(* Logix 5000 project; controller Leitura_AlfaInstrumentos_2711 vendor 1 type 14 code 149 rev 20.19; software revision 20.04 *)

TASK MainTask (continuous, watchdog 500 ms) : Balancas

MODULES
   Local : vendor 1 type 14 code 149 (Compact 0, rev 20.19)
      Discrete_IO : Embedded (Compact 1, rev 3.1, Output RPI 20 ms)
      BL04 : vendor 90 type 0 code 46 (Ethernet 192.168.1.53, rev 1.5, StandardDataDriven RPI 10 ms)
           BL04:I.DATA[5].1   // Unidade
           BL04:I.DATA[5].5   // 1 = Vazia
           BL04:I.DATA[5].0   // 1 = Erro
           BL04:I.DATA[15]   // Tara
           BL04:I.DATA[14]   // Tara
           BL04:I.DATA[13]   // Tara
           BL04:I.DATA[12]   // Tara
           BL04:I.DATA[5].2   // Unidade
           BL04:I.DATA[10]   // Peso Bruto ou Liquido
           BL04:I.DATA[8]   // Peso Bruto ou Liquido
           BL04:I.DATA[9]   // Peso Bruto ou Liquido
           BL04:I.DATA[11]   // Peso Bruto ou Liquido
           BL04:I.DATA[4].7   // 0 = Peso Bruto / 1 = Peso Liquido
           BL04:I.DATA[4].0   // Casas Decimais
           BL04:I.DATA[4].1   // Casas Decimais
           BL04:I.DATA[4].2   // Casas Decimais
           BL04:I.DATA[5].6   // 1 = Calibração
           BL04:I.DATA[4].5   // 1 = Saturação
           BL04:I.DATA[4].3   // 1= PesoNegativo
           BL04:I.DATA[4].4   // 1 = Variação do peso igual ou acima do valor configurado em MOV
           BL04:I.DATA[5].3   // 1 = Variação do peso igual ou acima do valor configurado em MOV
           BL04:I.DATA[5].4   // 1 = Tara Negativa
           BL04:I.DATA[4].6   // 1 = Sobrecarga
END_MODULES

VAR_GLOBAL   (* controller tags *)
   BL04_PesoBruto : REAL := 0.4;
   BL04_PesoOK : BOOL := 1;   // Indica que o peso é valido
END_VAR

PROGRAM Balancas   (* main routine Principal *)
VAR
   BL04_PesoDINT : DINT := 1053609165;
END_VAR

ROUTINE BL04   (* ladder *)
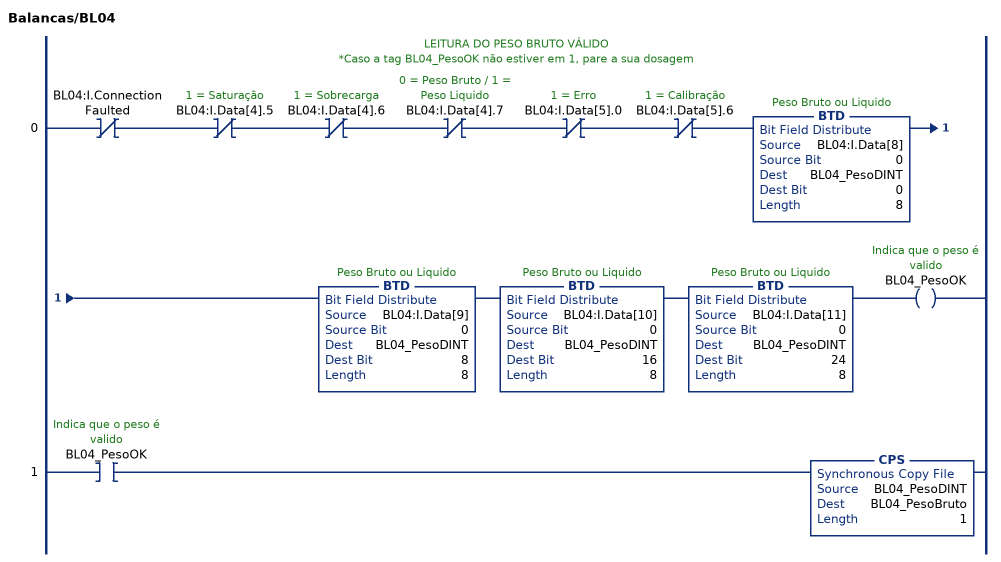
   // LEITURA DO PESO BRUTO VÁLIDO
   // *Caso a tag BL04_PesoOK não estiver em 1, pare a sua dosagem
   0: XIO(BL04:I.ConnectionFaulted)XIO(BL04:I.Data[4].5)XIO(BL04:I.Data[4].6)XIO(BL04:I.Data[4].7)XIO(BL04:I.Data[5].0)XIO(BL04:I.Data[5].6)BTD(BL04:I.Data[8],0,BL04_PesoDINT,0,8)BTD(BL04:I.Data[9],0,BL04_PesoDINT,8,8)BTD(BL04:I.Data[10],0,BL04_PesoDINT,16,8)BTD(BL04:I.Data[11],0,BL04_PesoDINT,24,8)OTE(BL04_PesoOK);
   1: XIC(BL04_PesoOK)CPS(BL04_PesoDINT,BL04_PesoBruto,1);
END_ROUTINE

ROUTINE Principal   (* ladder *)
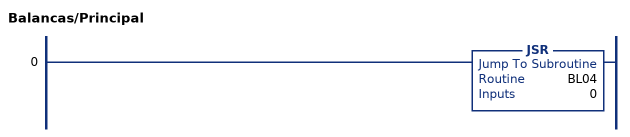
   0: JSR(BL04,0);
END_ROUTINE
END_PROGRAM
